// Mitsubishi GX Works2 project: PLC311122FINAL   PLC: FX3G

// global labels: Global1
VAR_GLOBAL
  Start_day_lamp AT Y010 : BOOL;  (* נורה שתישאר דלוקה עד סוף היום או שאחד התנאים של הפרת יום עבודה קורה *)
  Orange_tank AT D1100 : REAL;  (* קיבולת מיכל התפוזים *)
  Clementine_tank AT D1102 : REAL;  (* קיבולת מיכל הקלמטינות *)
  Pomelo_tank AT D1104 : REAL;  (* קיבולת מיכל הפומלות *)
  Orange_quantity AT D1106 : REAL;  (* ערך כמות של התפוזים *)
  Clementine_quantity AT D1108 : REAL;  (* ערך כמות של הקלמנטינות *)
  Pomelo_quantity AT D1110 : REAL;  (* ערך כמות של הפומלות *)
END_VAR
VAR_GLOBAL CONSTANT
  Constant_3_sec : INT := 30;  (* קבוע - 3 שניות *)
  Constant_5_sec : INT := 50;  (* קבוע - 5 שניות *)
  Constant_0 : REAL;  (* קבוע 0 *)
END_VAR
VAR_GLOBAL
  Timer_washing_fruits AT TC0 : BOOL;  (* טיימר - תחילת שלב שטיפת פירות *)
  Timer_washing_fruits_result AT TS0 : BOOL;  (* תוצאת הטיימר תחילת שלב שטיפת פירות *)
  Start_counting_x11_press AT CC0 : BOOL;  (* שם המונה הסופר את מספר הלחיצות על מתג להתחלת סחיטת הפירות *)
  Counter_x11_press_result AT CS0 : BOOL;  (* תוצאת המונה הסופר את מספר הלחיצות על מתג להתחלת סחיטת הפירות *)
  Counter_x3_press_result AT CS1 : BOOL;  (* תוצאת המונה הסופר את מספר הלחיצות על מתג להתחלת בדיקת איכות המיץ *)
  start_washing_fruits_button AT X002 : BOOL;  (* מתג התחלת שלב שטיפת פירות *)
  Transfer_to_squeez_tank_button AT X001 : BOOL;  (* מתג 1, איסוף הפירות *)
  start_fruits_squeez_button AT X011 : BOOL;  (* מתג 11, מתחיל את סחיטת הפירות *)
  start_calc_profit_from_juice AT X006 : BOOL;  (* מתג המציין את תחילת שלב הסעיף הפתוח - חישוב השווי הכספי של המיץ שיוצר באיטרציה ספציפית *)
  start_juice_quality_button AT X003 : BOOL;  (* מתג 3, מתחיל את בדיקת האיכות *)
  Start_day AT X010 : BOOL;  (* מתג תחילת יום עבודה *)
  SW_7_Emergenncy AT X007 : BOOL;  (* מתג 7 משמש למקרה חירום *)
  Fruits_moving_to_washing_machine AT Y005 : BOOL;  (* נורה שמעידה על התחלת שלב העברת הפירות ממיכלי המלאי למכונות השטיפה *)
  collecting_fruits_lamp AT Y001 : BOOL;  (* נורה שתשאר דלוקה לאורך שלב איסוף הפירות והעברה למיכל יעודי *)
  squeez_process_blink_lamp2 AT Y002 : BOOL;  (* נורה 2, תהבהב בזמן הסחיטה לסרוגין *)
  squeez_process_blink_lamp3 AT Y003 : BOOL;  (* נורה 3, תהבהב בזמן הסחיטה לסרוגין *)
  juice_quality_test_lamp AT Y004 : BOOL;  (* נורה 4, נדלקת ל5 שניות כאשר הבדיקה הצליחה (הערך האנלוגי בטווח) *)
  Juice_tank AT D1112 : REAL;  (* מיכל המיץ *)
  Washing_machine_orange AT D1114 : REAL;  (* מכונת שטיפה תפוזים *)
  Washing_machine_clementine AT D1116 : REAL;  (* מכונת שטיפה קלמטינות *)
  Washing_machine_pomelo AT D1118 : REAL;  (* מכונת שטיפה פומלות *)
  Squeeze_tank AT D1120 : REAL;  (* מיכל סחיטה של כלל הפירות *)
  Storage_tank AT D1122 : REAL;  (* מיכל אחסון של המיץ *)
  Orange_capacity_temp AT D1124 : REAL;  (* שומר את הערך המינימלי של כמות התפוזים בשלב העברה לשטיפה *)
  Pomelo_and_clementine_capacity AT D1126 : REAL;  (* כמות הקלמנטינות והפומלות שנכניס למיכלי השטיפה *)
  Orange_capacity_minimal AT D1128 : REAL;  (* שמירת הערך המינימלי של כמות התפוזים שצריך להעביר לשטיפה *)
  Analog_value AT D1130 : REAL;  (* הערך האנלוגי של הדגימה שיצאה *)
END_VAR
VAR_GLOBAL CONSTANT
  Constant_1 : REAL := 1;  (* קבוע 1 *)
  Constant_100 : REAL := 100;  (* קבוע 100 עבור כמות התפוזים המקסימלית במכונת השטיפה *)
  Constant_2 : REAL := 2;  (* קבוע 2 לחלוקת הכמות במכונת שטיפה *)
  Counter_2_presses : INT := 2;  (* מונה הסופר 2 לחיצות *)
  const_1_sec : INT := 10;  (* קבוע 1 שנייה *)
  Const_404_5 : REAL := 404.5;  (* קבוע- 404.5 להמרה בין הקלט האנלוגי לערכי הבקר *)
  Const_5 : REAL := 5;  (* קבוע 5 *)
END_VAR
VAR_GLOBAL
  Orange_minimal_split_indicator AT M104 : BOOL;  (* נורת דמה שמעידה שמצאנו ערך מינימלי לכמות התפוזים *)
  End_washing_orange AT M105 : BOOL;  (* נורת אינדיקציה שסיימנו את שלב שטיפת התפוזים *)
  End_washing_clementin AT M106 : BOOL;  (* נורת אינדיקציה שסיימנו את שלב שטיפת הקלמטינות *)
  End_washing_pomelo AT M107 : BOOL;  (* נורת אינדיקציה שסיימנו את שלב שטיפת הפומלות *)
  Start_transfer_squeez_process AT M108 : BOOL;  (* נורת אינדיקציה לתחילת שלב העברת הפירות ממכונת השטיפה למכונת הסחיטה *)
  End_transfer_squeez_process AT M109 : BOOL;  (* נורת אינדיקציה לסוף שלב העברת הפירות ממכונת השטיפה למכונת הסחיטה *)
  End_transfer_to_squeez_tank AT M110 : BOOL;  (* נורת עזר לסיום העברת הפירות למיכל הסחיטה *)
  Start_washing_fruits_process AT M111 : BOOL;  (* נורת עזר המציינת את התחלת שלב העברת הפירות ממכלי הפירות למכונות השטיפה *)
  Start_blinking AT M112 : BOOL;  (* נורת עזר להבהוב *)
  help_blinking AT M113 : BOOL;  (* משתנה עזר להבהוב *)
  End_of_squeez AT M114 : BOOL;  (* נורת עזר - סיום סחיטה והתחלת העברת הפירות הסחוטים למיכל המיץ *)
  End_trasfer_to_juice_tank AT M115 : BOOL;  (* נורת עזר - סיום העברה למיכל המיץ *)
  Check_min_value AT M116 : BOOL;  (* נורה שתצביע כי נבחר יותר מ1 בכניסה האנלוגית *)
  Check_max_value AT M117 : BOOL;  (* נורה שתצביע כי נבחר פחות מ5 בכניסה האנלוגית *)
  Analog_check_correct AT M118 : BOOL;  (* נורה שמצביעה כי הטווח בקלט האנלוגי תקין *)
  The_juice_not_good AT M119 : BOOL;  (* נורת עזר שמעידה שצריך לזרוק את המיץ באיטרציה זו מחשש לבקטריות *)
  Fill_storage_tank AT M120 : BOOL;  (* נורת אינדיקציה למילוי מיכל האחסון *)
  Threw_the_juice AT M121 : BOOL;  (* נורת אינדיקציה לזריקת המיץ לאחר 2 בדיקות עם ערך לא תקין *)
  End_day AT M122 : BOOL;  (* נורת סיום יום לאחר לחיצה על מתג 7 *)
  Not_enough_stock AT M123 : BOOL;  (* נורת אינדיקציה שאין מספיק מלאי לאחד הפירות *)
  Blinking_end_day AT M124 : BOOL;  (* נורת עזר להיבהוב סוף יום *)
  Blinking_end_day_Help AT M125 : BOOL;  (* נורת עזר להיבהוב *)
  Help_blink_lamp_10 AT M126 : BOOL;  (* נורת עזר להבהוב סוף יום של נורה 10 *)
  end_transfer_or_not_to_storage AT M128 : BOOL;  (* נורת עזר לסיום שלב בדיקת איכות המיץ והעברה או אי העברה של המיץ למיכל האחסון *)
  Timer_blinking_input_lamp_2 AT TC1 : BOOL;  (* מונה טיימר של y2 *)
  Timer_blinking_input_lamp_3 AT TC2 : BOOL;  (* מונה טיימר של y3 *)
  Timer_squeez_time AT TC3 : BOOL;  (* מונה טיימר 3 שניות *)
  Timer_juice_quality AT TC4 : BOOL;  (* מונה טיימר 5 שניות *)
  Timer_end_day_3_sec AT TC5 : BOOL;  (* מונה טיימר 3 שניות לסיום יום *)
  Timer_blink_end_day AT TC6 : BOOL;  (* מונה היבהוב סוף יום *)
  Timer_blinking_lamp_2_result AT TS1 : BOOL;  (* מונה טיימר של תוצאה y2 *)
  Timer_blinking_lamp_3_result AT TS2 : BOOL;  (* מונה טיימר של תוצאה y3 *)
  Timer_squeez_time_result AT TS3 : BOOL;  (* תוצאת מונה טיימר 3 שניות *)
  Timer_juice_quality_result AT TS4 : BOOL;  (* תוצאת מונה טיימר 5 שניות *)
  End_day_3_sec_result AT TS5 : BOOL;  (* תוצאה של TC5 *)
  Timer_blink_end_day_result AT TS6 : BOOL;  (* תוצאת מונה היבהוב סוף יום *)
  Start_counting_x3_press AT CC1 : BOOL;  (* שם המונה הסופר את מספר הלחיצות על מתג להתחלת בדיקת איכות המיץ *)
  juice_tank_help_calc_profit AT D1132 : REAL;  (* רגיסטר עזר למיכל המיץ אשר עוזר חשב את השווי הכספי מהמיץ שנוצר באיטרציה ספציפית *)
  total_profit_from_juice AT D8282 : INT;  (* רגיסטר תצוגה אנלוגית אשר מציג את הרווח פר איטרציה מכמות המיץ שנוצר *)
  Analog_juice_quality AT D8281 : INT;  (* קלט אנלוגי שבודק את איכות המיץ *)
  end_calc_profit_analog_output AT M129 : BOOL;  (* נורת עזר שמעידה שהסתיים חישוב שווי הרווח ממיץ באיטרציה ספציפית אשר השווי גדול מ - 0 *)
  Timer_calc_profit_from_juice AT TC7 : BOOL;  (* מונה זמן שעובד בזמן שמחשבים את השווי רווח של המיץ שנוצר באיטרציה ספציפית *)
  Calc_profit_from_juice_result AT TS7 : BOOL;  (* תוצאת מונה זמן שעובד בזמן שמחשבים את השווי רווח של המיץ שנוצר באיטרציה ספציפית *)
  Profit_from_juice_lamp AT Y006 : BOOL;  (* נורה שתשאר דלוקה 3 שניות בעת חישוב הרווח מהמיץ שנוצר באיטרציה ספציפית *)
END_VAR
VAR_GLOBAL CONSTANT
  money_value_per_liter : REAL := 0.0717;  (* קבוע אשר מציין את שווי המיץ באיטרציה מסויימת פר ליטר *)
END_VAR
VAR_GLOBAL
  Timer_blink_end_day_2 AT TC8 : BOOL;  (* מונה הבהוב סוף יום *)
  Timer_blink_end_day_result_2 AT TS8 : BOOL;  (* תוצאת מונה טיימר הבהוב סוף יום *)
  Help_blink_lamp_10_temp AT M130 : BOOL;  (* נורת עזר להבהוב סוף יום *)
END_VAR
VAR_GLOBAL CONSTANT
  const_half_sec : INT := 5;
END_VAR
VAR_GLOBAL
  not_valid_quantities_of_fruits AT M127 : BOOL;  (* נורת עזר לבדיקת מקרה קיצון שהזנת הקלט של כמות התפוזים גדולה מ - 0 ובדיקת תנאי תחילת יום עבודה *)
  check_quantities_of_fruits AT M131 : BOOL;  (* נורת עזר שבודקת עם הקלט בעצם תקין של הפירות *)
  end_day_INDICATOR AT M132 : BOOL;  (* נורת עזר להיבהוב סוף יום *)
  start_day_indicator AT M133 : BOOL;  (* נורת עזר לאינדיקציה אם אנחנו בעצם יכולים להתחיל את היום *)
END_VAR

// task Task_01 (event TRUE, interval 0, priority 31): POU_01

PROGRAM POU_01
(* structured ladder/FBD written out as ST: instructions are called as NAME(EN, inputs, outputs); _pN, _eN, _tN stand for wires *)
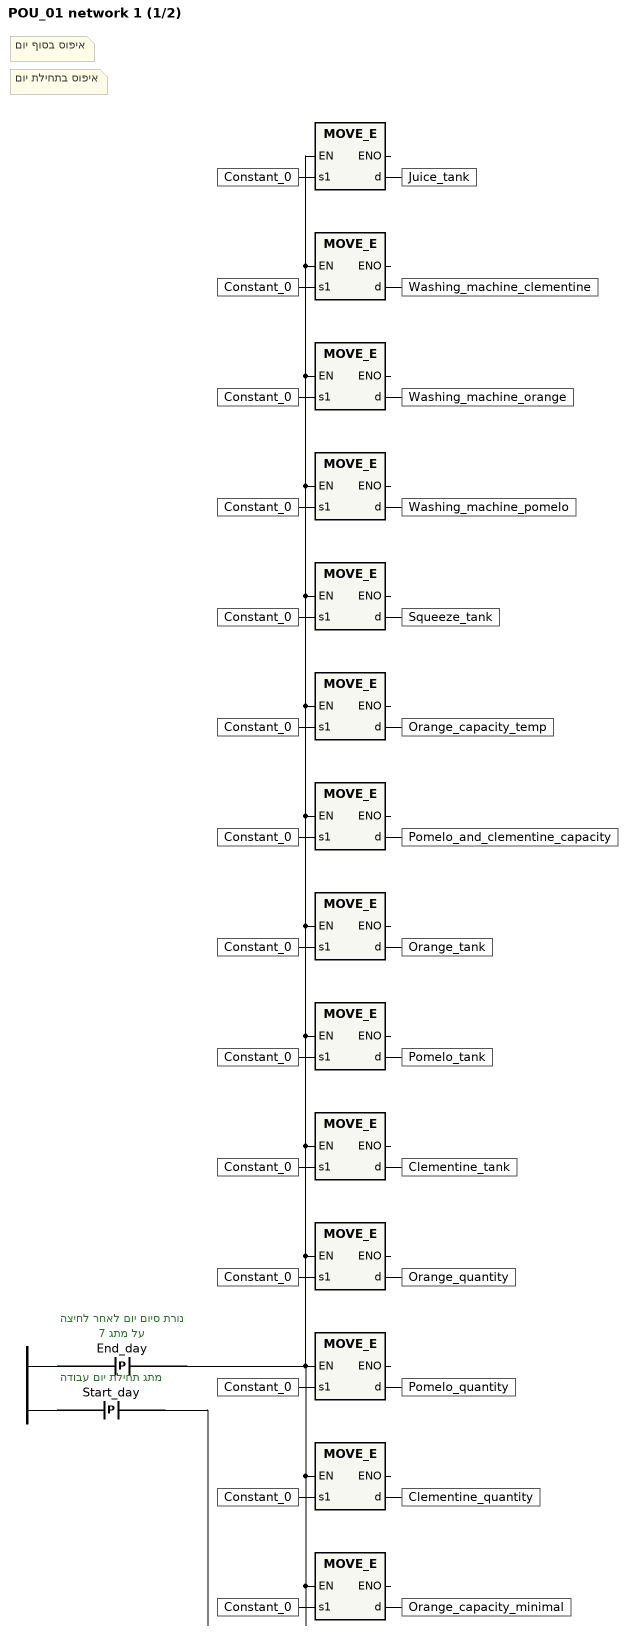
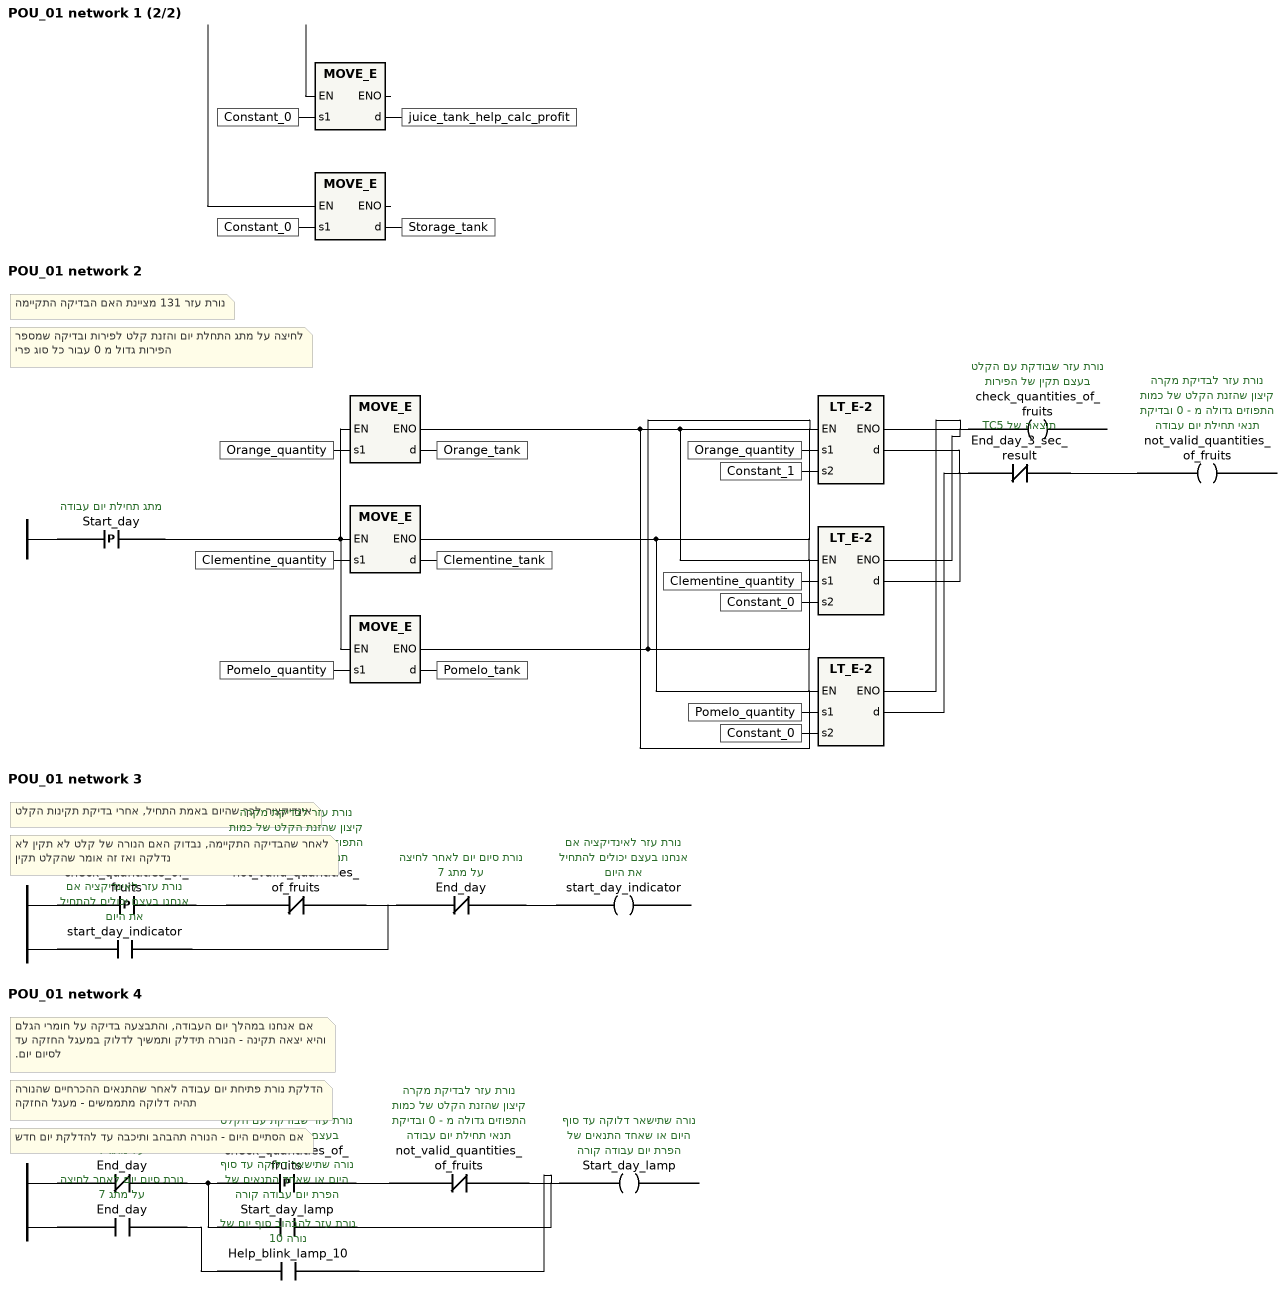
(* network 1 *)
(* איפוס בסוף יום *)
(* איפוס בתחילת יום *)
_p1 := LDP(TRUE, End_day);
MOVE_E(_p1, Constant_0, Juice_tank);
MOVE_E(_p1, Constant_0, Washing_machine_clementine);
MOVE_E(_p1, Constant_0, Washing_machine_orange);
MOVE_E(_p1, Constant_0, Washing_machine_pomelo);
MOVE_E(_p1, Constant_0, Squeeze_tank);
MOVE_E(_p1, Constant_0, Orange_capacity_temp);
MOVE_E(_p1, Constant_0, Pomelo_and_clementine_capacity);
MOVE_E(_p1, Constant_0, Orange_tank);
MOVE_E(_p1, Constant_0, Pomelo_tank);
MOVE_E(_p1, Constant_0, Clementine_tank);
MOVE_E(_p1, Constant_0, Orange_quantity);
MOVE_E(_p1, Constant_0, Pomelo_quantity);
MOVE_E(_p1, Constant_0, Clementine_quantity);
MOVE_E(_p1, Constant_0, Orange_capacity_minimal);
MOVE_E(_p1, Constant_0, juice_tank_help_calc_profit);
MOVE_E(LDP(TRUE, Start_day), Constant_0, Storage_tank);
(* network 2 *)
(* נורת עזר 131 מציינת האם הבדיקה התקיימה *)
(* לחיצה על מתג התחלת יום והזנת קלט לפירות ובדיקה שמספר הפירות גדול מ 0 עבור כל סוג פרי *)
_p1 := LDP(TRUE, Start_day);
_e2 := MOVE_E(_p1, Orange_quantity, Orange_tank);
_e3 := MOVE_E(_p1, Clementine_quantity, Clementine_tank);
_e4 := MOVE_E(_p1, Pomelo_quantity, Pomelo_tank);
_p5 := _e2 OR _e3 OR _e4;
_e7 := LT_E(_p5, Orange_quantity, Constant_1, _t6);
_e9 := LT_E(_p5, Clementine_quantity, Constant_0, _t8);
_e11 := LT_E(_p5, Pomelo_quantity, Constant_0, _t10);
check_quantities_of_fruits := _e7 OR _e9 OR _e11;
not_valid_quantities_of_fruits := (_t6 OR _t8 OR _t10) AND NOT End_day_3_sec_result;
(* network 3 *)
(* אינדיקציה לכך שהיום באמת התחיל, אחרי בדיקת תקינות הקלט *)
(* לאחר שהבדיקה התקיימה, נבדוק האם הנורה של קלט לא תקין לא נדלקה ואז זה אומר שהקלט תקין *)
start_day_indicator := ((LDP(TRUE, check_quantities_of_fruits) AND NOT not_valid_quantities_of_fruits) OR start_day_indicator) AND NOT End_day;
(* network 4 *)
(* אם אנחנו במהלך יום העבודה, והתבצעה בדיקה על חומרי הגלם והיא יצאה תקינה - הנורה תידלק ותמשיך לדלוק במעגל החזקה עד לסיום יום. *)
(* הדלקת נורת פתיחת יום עבודה לאחר שהתנאים ההכרחיים שהנורה תהיה דלוקה מתממשים - מעגל החזקה *)
(* אם הסתיים היום - הנורה תהבהב ותיכבה עד להדלקת יום חדש *)
_p1 := NOT End_day;
Start_day_lamp := (_p1 AND LDP(TRUE, check_quantities_of_fruits) AND NOT not_valid_quantities_of_fruits) OR (_p1 AND Start_day_lamp) OR (End_day AND Help_blink_lamp_10);
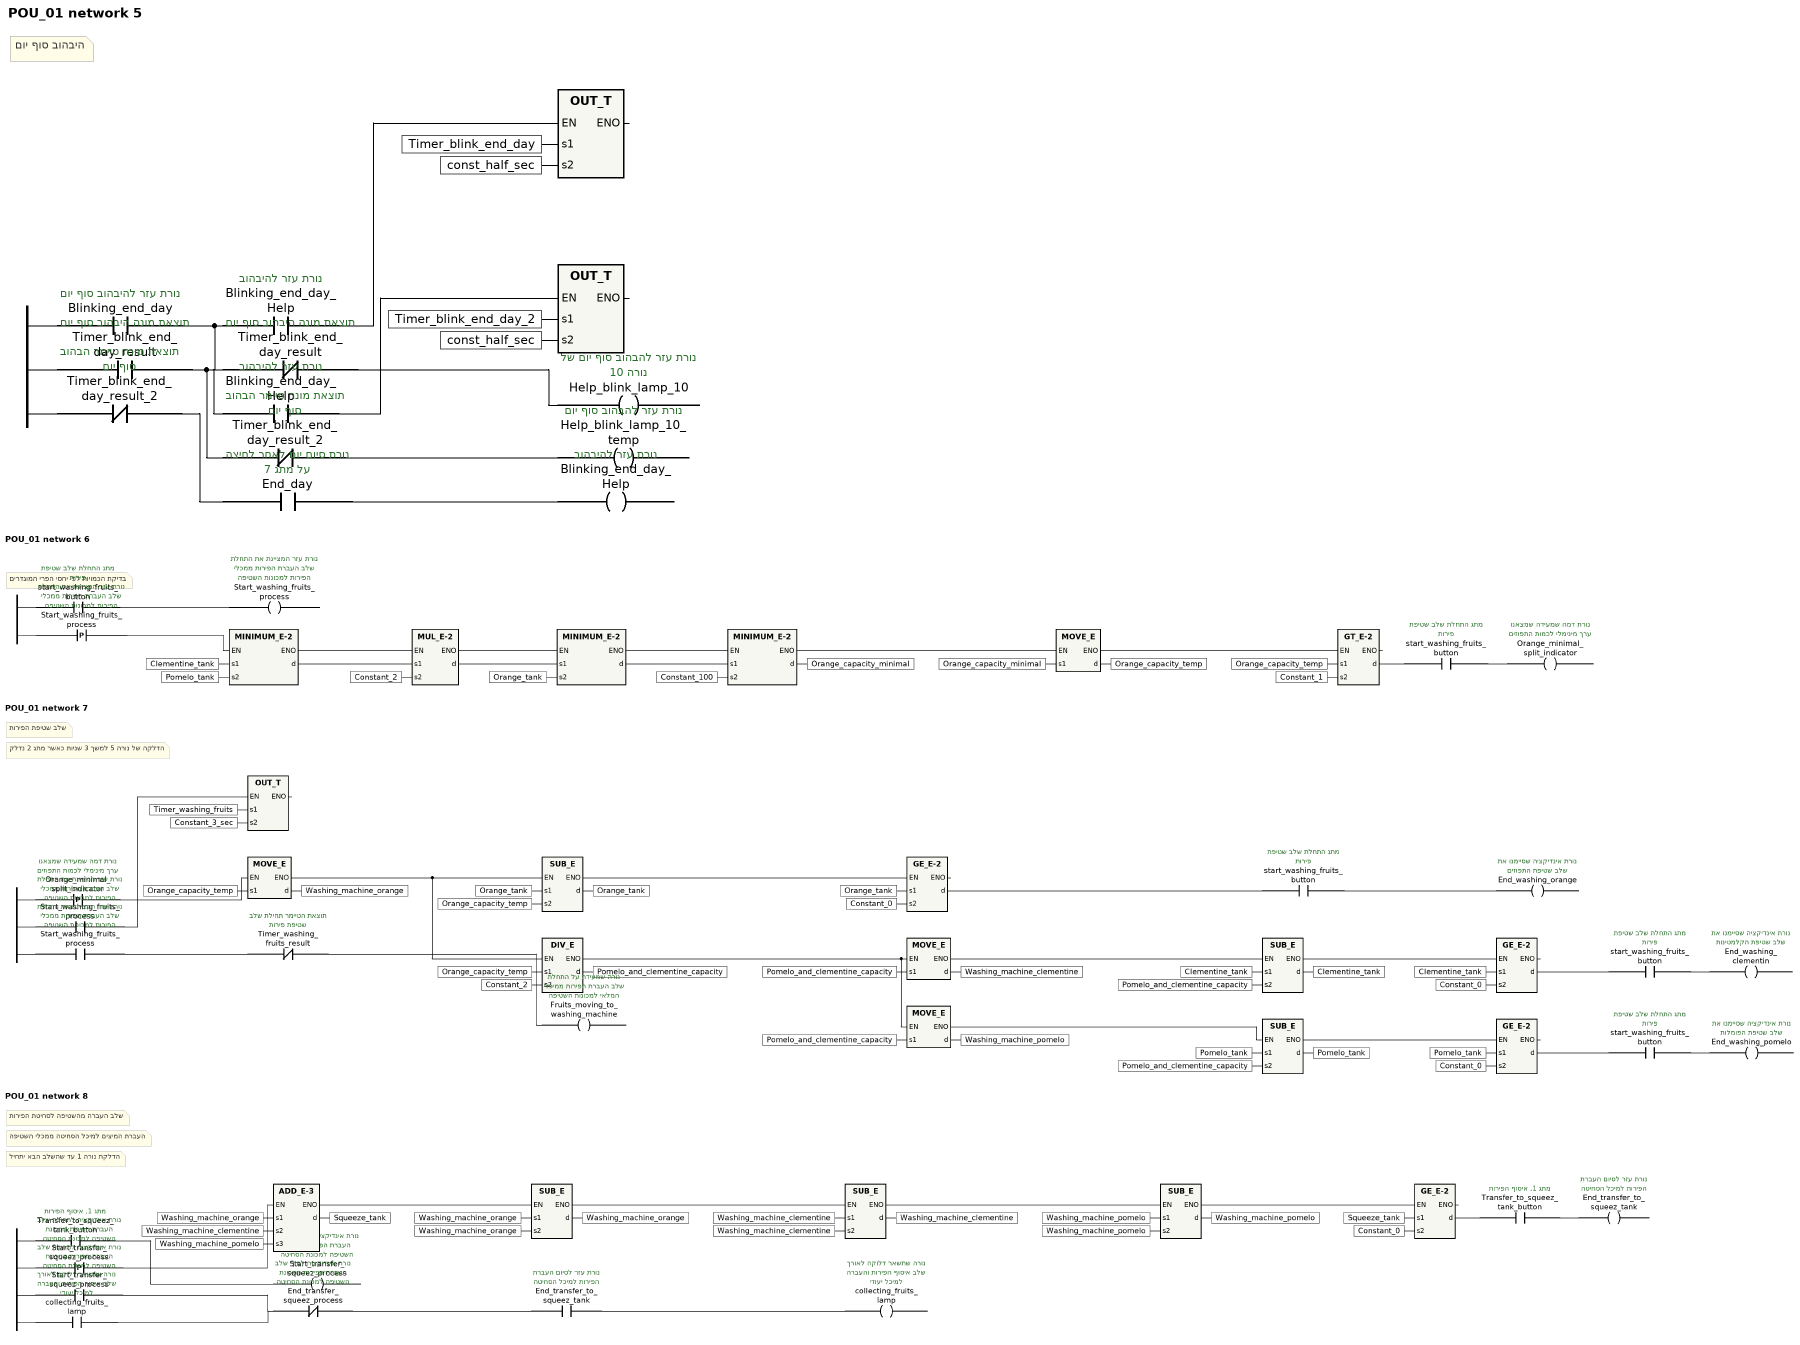
(* network 5 *)
(* היבהוב סוף יום *)
OUT_T(Blinking_end_day AND Blinking_end_day_Help, Timer_blink_end_day, const_half_sec);
Help_blink_lamp_10 := Blinking_end_day AND NOT Timer_blink_end_day_result;
OUT_T(Timer_blink_end_day_result AND Blinking_end_day_Help, Timer_blink_end_day_2, const_half_sec);
Help_blink_lamp_10_temp := Timer_blink_end_day_result AND NOT Timer_blink_end_day_result_2;
Blinking_end_day_Help := NOT Timer_blink_end_day_result_2 AND End_day;
(* network 6 *)
(* בדיקת הכמויות לפי יחסי הפרי המוגדרים *)
Start_washing_fruits_process := start_washing_fruits_button;
_e2 := MINIMUM_E(LDP(TRUE, Start_washing_fruits_process), Clementine_tank, Pomelo_tank, _t1);
_e4 := MUL_E(_e2, _t1, Constant_2, _t3);
_e6 := MINIMUM_E(_e4, _t3, Orange_tank, _t5);
_e7 := MINIMUM_E(_e6, _t5, Constant_100, Orange_capacity_minimal);
_e8 := MOVE_E(_e7, Orange_capacity_minimal, Orange_capacity_temp);
GT_E(_e8, Orange_capacity_temp, Constant_1, _t9);
Orange_minimal_split_indicator := _t9 AND start_washing_fruits_button;
(* network 7 *)
(* שלב שטיפת הפירות *)
(* הדלקה של נורה 5 למשך 3 שניות כאשר מתג 2 נדלק *)
_e1 := MOVE_E(LDP(TRUE, Orange_minimal_split_indicator), Orange_capacity_temp, Washing_machine_orange);
_e2 := SUB_E(_e1, Orange_tank, Orange_capacity_temp, Orange_tank);
GE_E(_e2, Orange_tank, Constant_0, _t3);
End_washing_orange := _t3 AND start_washing_fruits_button;
_e4 := DIV_E(_e1, Orange_capacity_temp, Constant_2, Pomelo_and_clementine_capacity);
_e5 := MOVE_E(_e4, Pomelo_and_clementine_capacity, Washing_machine_clementine);
_e6 := SUB_E(_e5, Clementine_tank, Pomelo_and_clementine_capacity, Clementine_tank);
GE_E(_e6, Clementine_tank, Constant_0, _t7);
End_washing_clementin := _t7 AND start_washing_fruits_button;
_e8 := MOVE_E(_e4, Pomelo_and_clementine_capacity, Washing_machine_pomelo);
_e9 := SUB_E(_e8, Pomelo_tank, Pomelo_and_clementine_capacity, Pomelo_tank);
GE_E(_e9, Pomelo_tank, Constant_0, _t10);
End_washing_pomelo := _t10 AND start_washing_fruits_button;
OUT_T(Start_washing_fruits_process, Timer_washing_fruits, Constant_3_sec);
Fruits_moving_to_washing_machine := Start_washing_fruits_process AND NOT Timer_washing_fruits_result;
(* network 8 *)
(* שלב העברה מהשטיפה לסחיטת הפירות *)
(* העברת המיצים למיכל הסחיטה ממכלי השטיפה *)
(* הדלקת נורה 1 עד שהשלב הבא יתחיל *)
Start_transfer_squeez_process := Transfer_to_squeez_tank_button;
_e1 := ADD_E(LDP(TRUE, Start_transfer_squeez_process), Washing_machine_orange, Washing_machine_clementine, Washing_machine_pomelo, Squeeze_tank);
_e2 := SUB_E(_e1, Washing_machine_orange, Washing_machine_orange, Washing_machine_orange);
_e3 := SUB_E(_e2, Washing_machine_clementine, Washing_machine_clementine, Washing_machine_clementine);
_e4 := SUB_E(_e3, Washing_machine_pomelo, Washing_machine_pomelo, Washing_machine_pomelo);
GE_E(_e4, Squeeze_tank, Constant_0, _t5);
End_transfer_to_squeez_tank := _t5 AND Transfer_to_squeez_tank_button;
collecting_fruits_lamp := ((Start_transfer_squeez_process OR collecting_fruits_lamp) AND NOT End_transfer_squeez_process) AND End_transfer_to_squeez_tank;
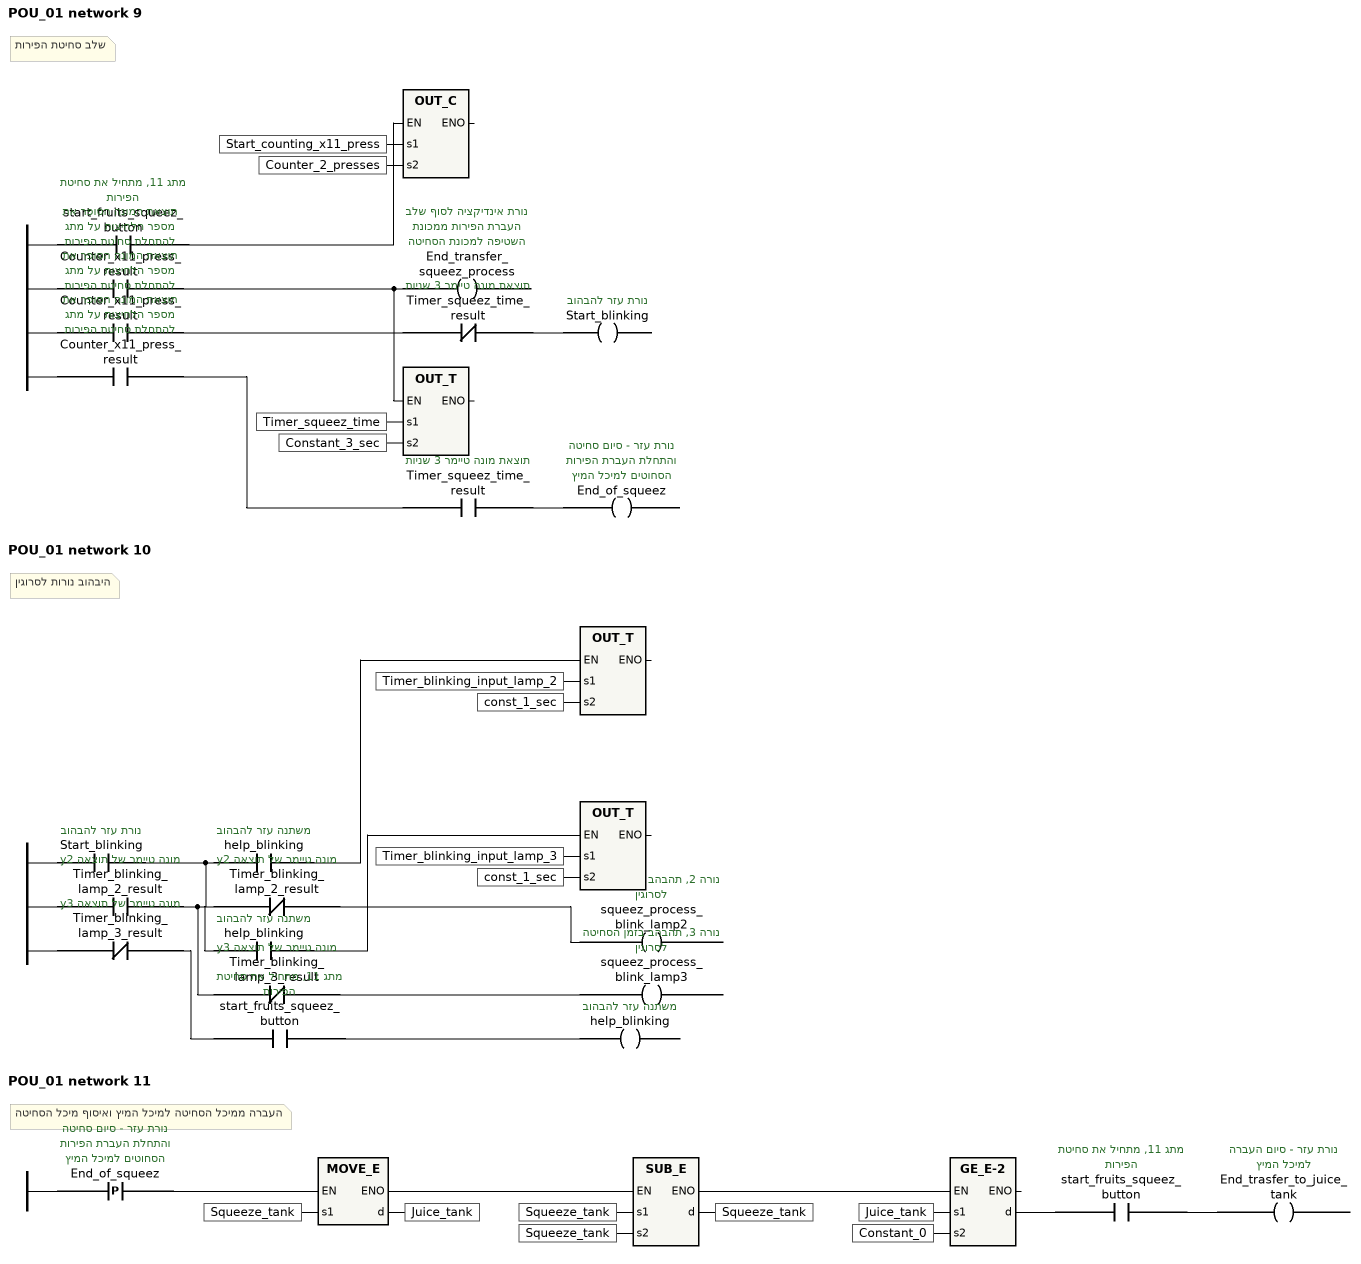
(* network 9 *)
(* שלב סחיטת הפירות *)
OUT_C(start_fruits_squeez_button, Start_counting_x11_press, Counter_2_presses);
End_transfer_squeez_process := Counter_x11_press_result;
OUT_T(Counter_x11_press_result, Timer_squeez_time, Constant_3_sec);
Start_blinking := Counter_x11_press_result AND NOT Timer_squeez_time_result;
End_of_squeez := Counter_x11_press_result AND Timer_squeez_time_result;
(* network 10 *)
(* היבהוב נורות לסרוגין *)
OUT_T(Start_blinking AND help_blinking, Timer_blinking_input_lamp_2, const_1_sec);
squeez_process_blink_lamp2 := Start_blinking AND NOT Timer_blinking_lamp_2_result;
OUT_T(Timer_blinking_lamp_2_result AND help_blinking, Timer_blinking_input_lamp_3, const_1_sec);
squeez_process_blink_lamp3 := Timer_blinking_lamp_2_result AND NOT Timer_blinking_lamp_3_result;
help_blinking := NOT Timer_blinking_lamp_3_result AND start_fruits_squeez_button;
(* network 11 *)
(* העברה ממיכל הסחיטה למיכל המיץ ואיסוף מיכל הסחיטה *)
_e1 := MOVE_E(LDP(TRUE, End_of_squeez), Squeeze_tank, Juice_tank);
_e2 := SUB_E(_e1, Squeeze_tank, Squeeze_tank, Squeeze_tank);
GE_E(_e2, Juice_tank, Constant_0, _t3);
End_trasfer_to_juice_tank := _t3 AND start_fruits_squeez_button;
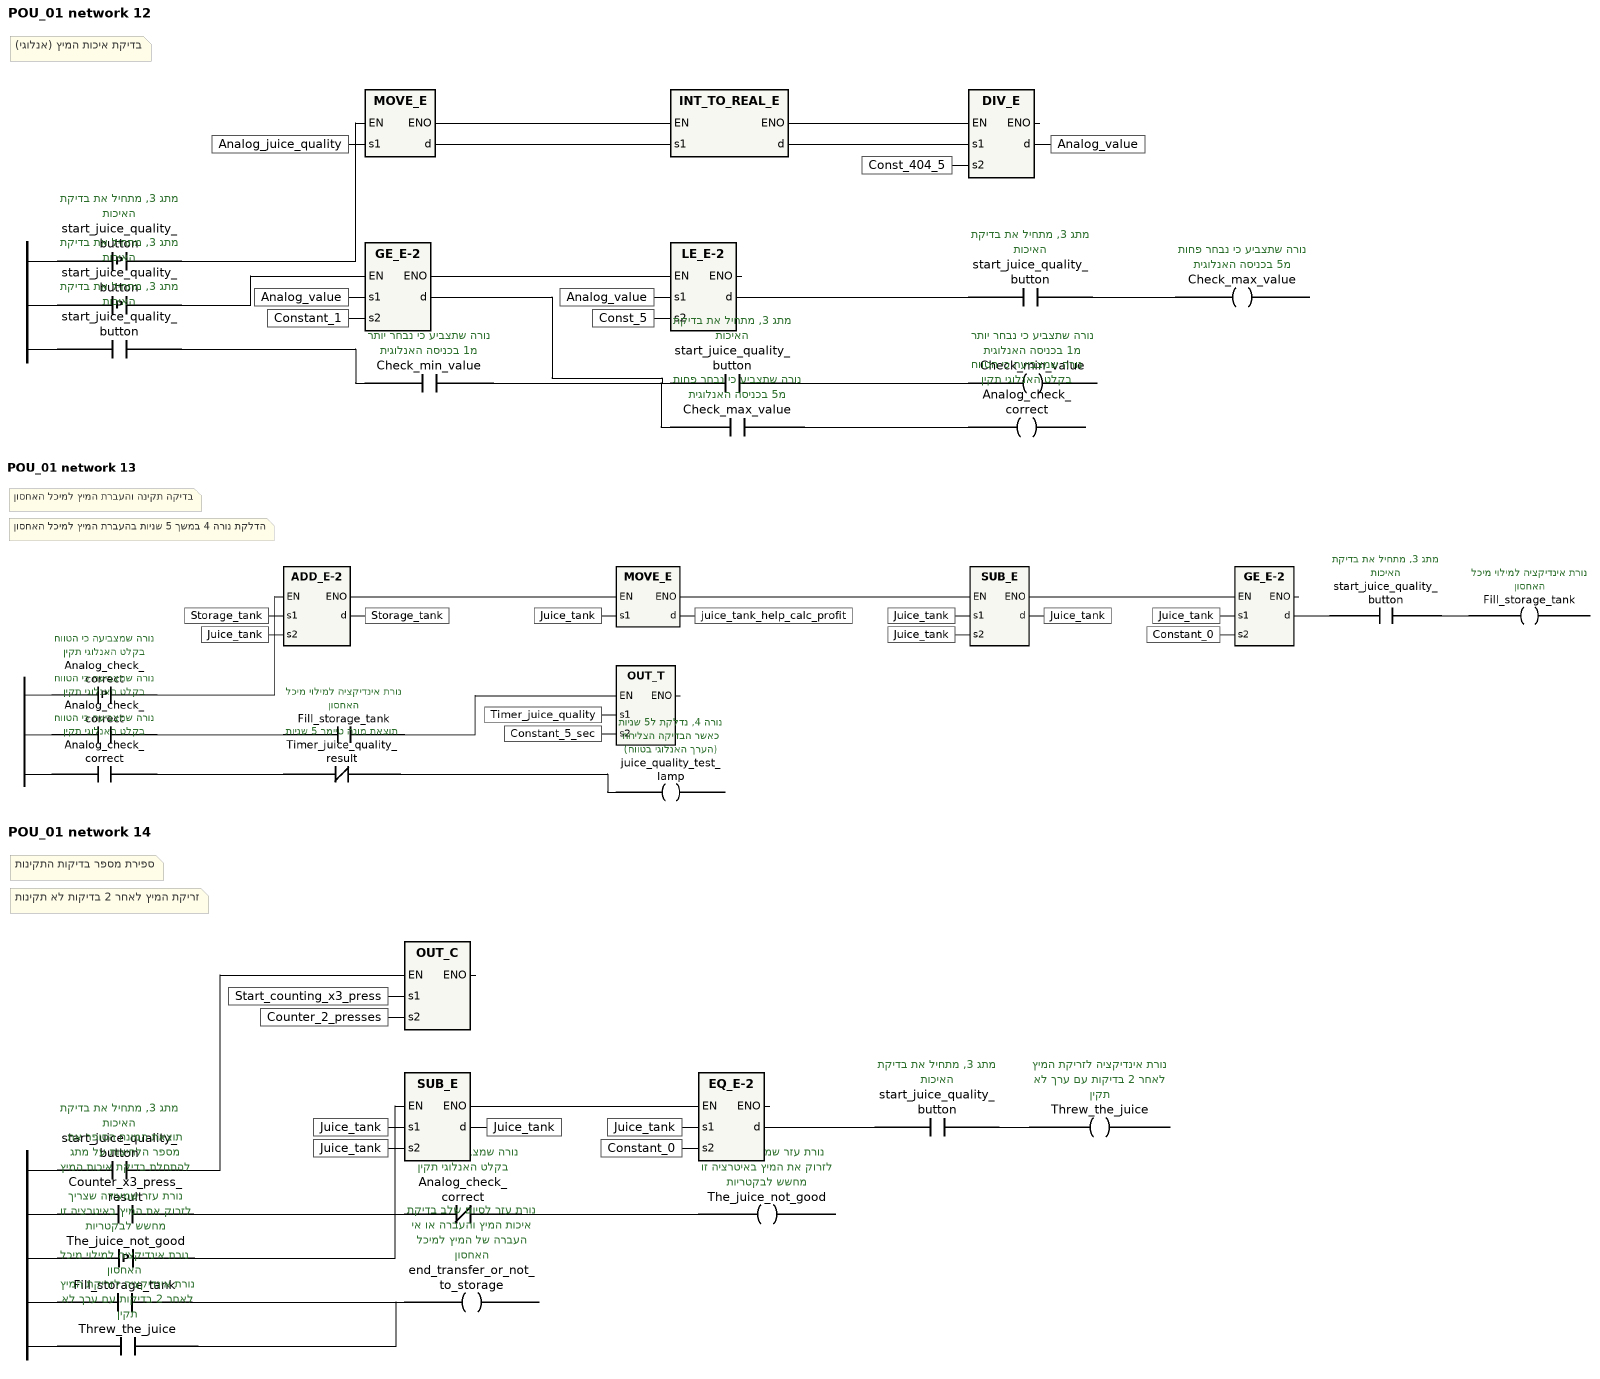
(* network 12 *)
(* בדיקת איכות המיץ (אנלוגי) *)
_e2 := MOVE_E(LDP(TRUE, start_juice_quality_button), Analog_juice_quality, _t1);
_e4 := INT_TO_REAL_E(_e2, _t1, _t3);
DIV_E(_e4, _t3, Const_404_5, Analog_value);
_e6 := GE_E(LDP(TRUE, start_juice_quality_button), Analog_value, Constant_1, _t5);
LE_E(_e6, Analog_value, Const_5, _t7);
Check_max_value := _t7 AND start_juice_quality_button;
Check_min_value := _t5 AND start_juice_quality_button;
Analog_check_correct := start_juice_quality_button AND Check_min_value AND Check_max_value;
(* network 13 *)
(* בדיקה תקינה והעברת המיץ למיכל האחסון *)
(* הדלקת נורה 4 במשך 5 שניות בהעברת המיץ למיכל האחסון *)
_e1 := ADD_E(LDP(TRUE, Analog_check_correct), Storage_tank, Juice_tank, Storage_tank);
_e2 := MOVE_E(_e1, Juice_tank, juice_tank_help_calc_profit);
_e3 := SUB_E(_e2, Juice_tank, Juice_tank, Juice_tank);
GE_E(_e3, Juice_tank, Constant_0, _t4);
Fill_storage_tank := _t4 AND start_juice_quality_button;
OUT_T(Analog_check_correct AND Fill_storage_tank, Timer_juice_quality, Constant_5_sec);
juice_quality_test_lamp := Analog_check_correct AND NOT Timer_juice_quality_result;
(* network 14 *)
(* ספירת מספר בדיקות התקינות *)
(* זריקת המיץ לאחר 2 בדיקות לא תקינות *)
OUT_C(start_juice_quality_button, Start_counting_x3_press, Counter_2_presses);
The_juice_not_good := Counter_x3_press_result AND NOT Analog_check_correct;
_e1 := SUB_E(LDP(TRUE, The_juice_not_good), Juice_tank, Juice_tank, Juice_tank);
EQ_E(_e1, Juice_tank, Constant_0, _t2);
Threw_the_juice := _t2 AND start_juice_quality_button;
end_transfer_or_not_to_storage := Fill_storage_tank OR Threw_the_juice;
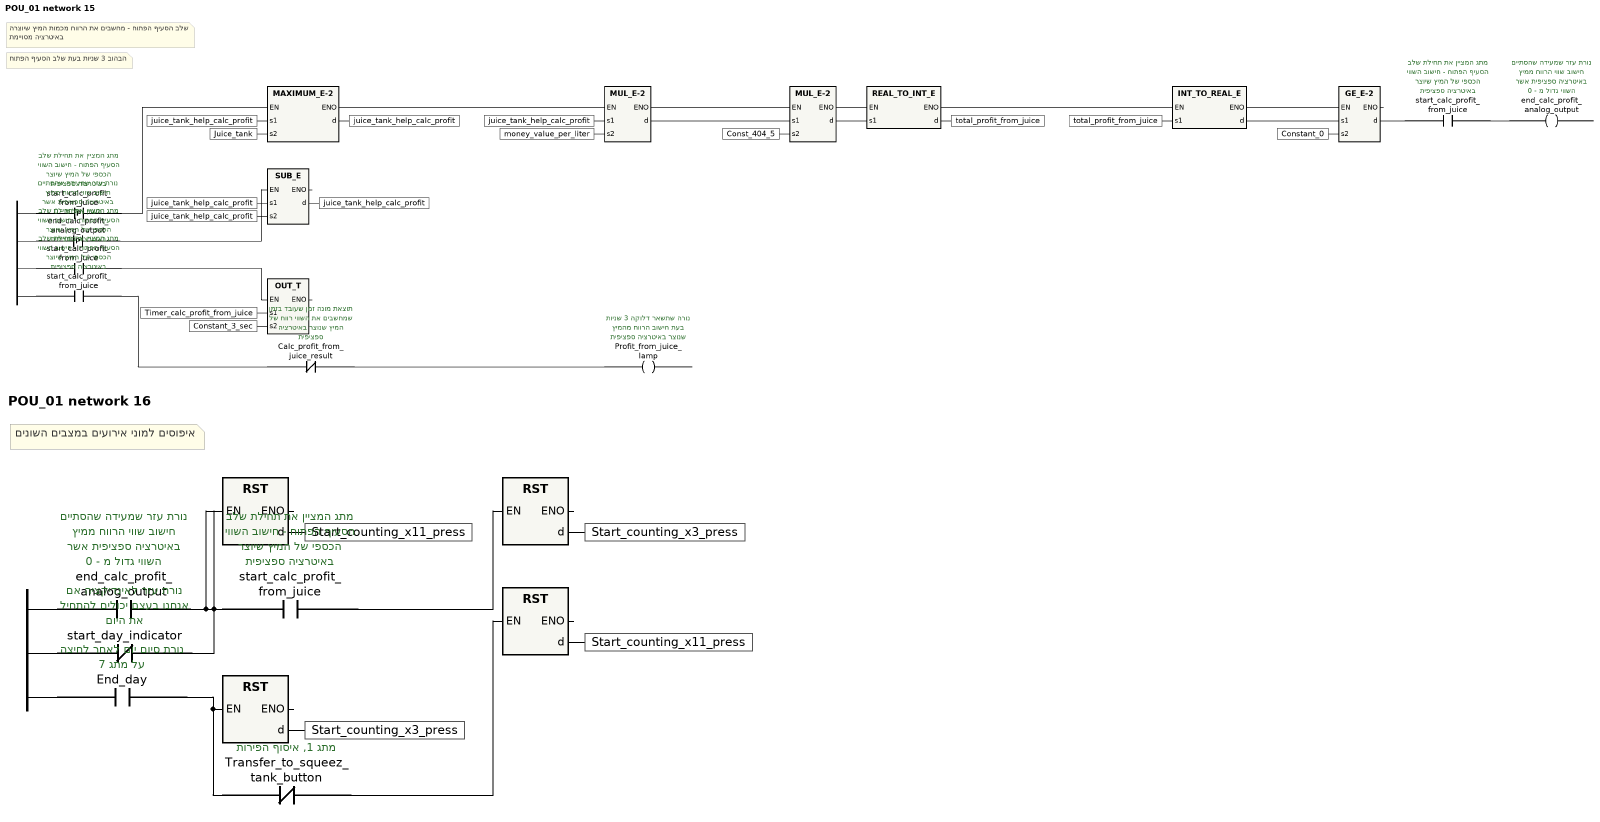
(* network 15 *)
(* שלב הסעיף הפתוח - מחשבים את הרווח מכמות המיץ שיוצרה באיטרציה מסויימת *)
(* הבהוב 3 שניות בעת שלב הסעיף הפתוח *)
_e1 := MAXIMUM_E(LDP(TRUE, start_calc_profit_from_juice), juice_tank_help_calc_profit, Juice_tank, juice_tank_help_calc_profit);
_e3 := MUL_E(_e1, juice_tank_help_calc_profit, money_value_per_liter, _t2);
_e5 := MUL_E(_e3, _t2, Const_404_5, _t4);
_e6 := REAL_TO_INT_E(_e5, _t4, total_profit_from_juice);
_e8 := INT_TO_REAL_E(_e6, total_profit_from_juice, _t7);
SUB_E(LDP(TRUE, end_calc_profit_analog_output), juice_tank_help_calc_profit, juice_tank_help_calc_profit, juice_tank_help_calc_profit);
GE_E(_e8, _t7, Constant_0, _t9);
end_calc_profit_analog_output := _t9 AND start_calc_profit_from_juice;
OUT_T(start_calc_profit_from_juice, Timer_calc_profit_from_juice, Constant_3_sec);
Profit_from_juice_lamp := start_calc_profit_from_juice AND NOT Calc_profit_from_juice_result;
(* network 16 *)
(* איפוסים למוני אירועים במצבים השונים *)
_p1 := end_calc_profit_analog_output OR (NOT start_day_indicator);
RST(_p1, Start_counting_x11_press);
RST(_p1 AND start_calc_profit_from_juice, Start_counting_x3_press);
RST(End_day AND NOT Transfer_to_squeez_tank_button, Start_counting_x11_press);
RST(End_day, Start_counting_x3_press);
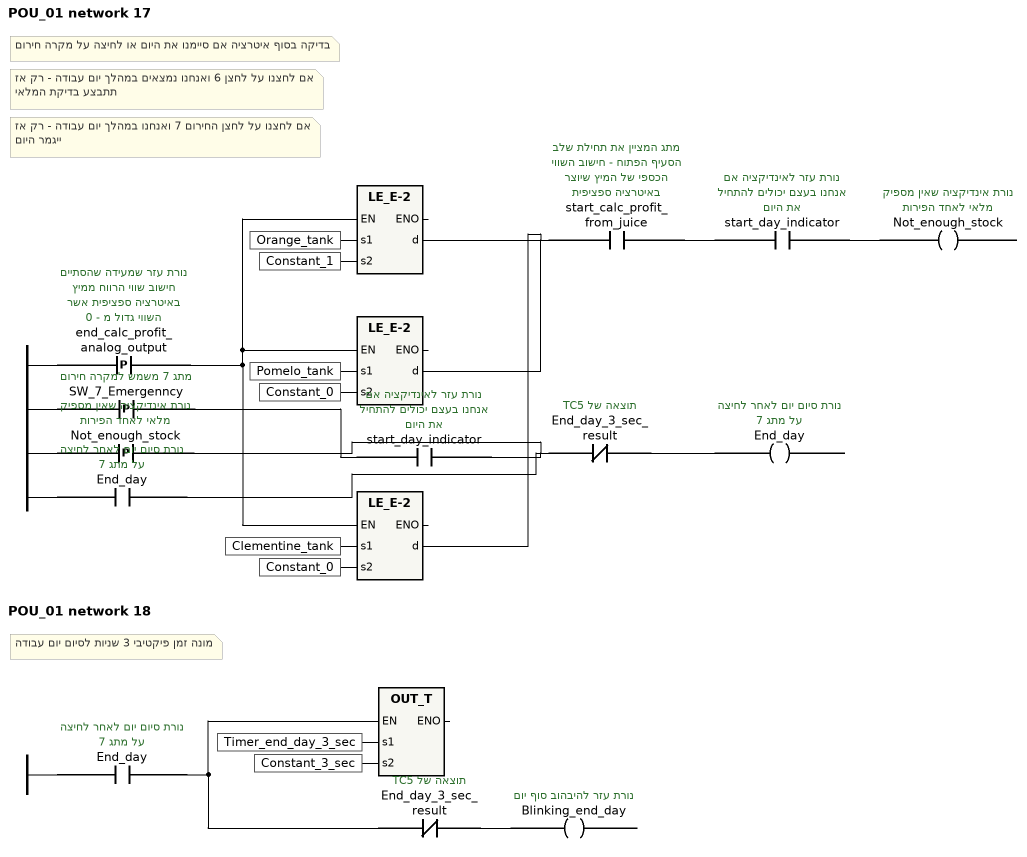
(* network 17 *)
(* בדיקה בסוף איטרציה אם סיימנו את היום או לחיצה על מקרה חירום *)
(* אם לחצנו על לחצן 6 ואנחנו נמצאים במהלך יום עבודה - רק אז תתבצע בדיקת המלאי *)
(* אם לחצנו על לחצן החירום 7 ואנחנו במהלך יום עבודה - רק אז ייגמר היום *)
_p1 := LDP(TRUE, end_calc_profit_analog_output);
LE_E(_p1, Orange_tank, Constant_1, _t2);
LE_E(_p1, Pomelo_tank, Constant_0, _t3);
LE_E(_p1, Clementine_tank, Constant_0, _t4);
Not_enough_stock := ((_t2 OR _t3 OR _t4) AND start_calc_profit_from_juice) AND start_day_indicator;
End_day := ((LDP(TRUE, SW_7_Emergenncy) AND start_day_indicator) OR LDP(TRUE, Not_enough_stock) OR End_day) AND NOT End_day_3_sec_result;
(* network 18 *)
(* מונה זמן פיקטיבי 3 שניות לסיום יום עבודה *)
OUT_T(End_day, Timer_end_day_3_sec, Constant_3_sec);
Blinking_end_day := End_day AND NOT End_day_3_sec_result;
END_PROGRAM
